// Mitsubishi GX Works2 project: main   PLC: FX3U/FX3UC

PROGRAM MAIN
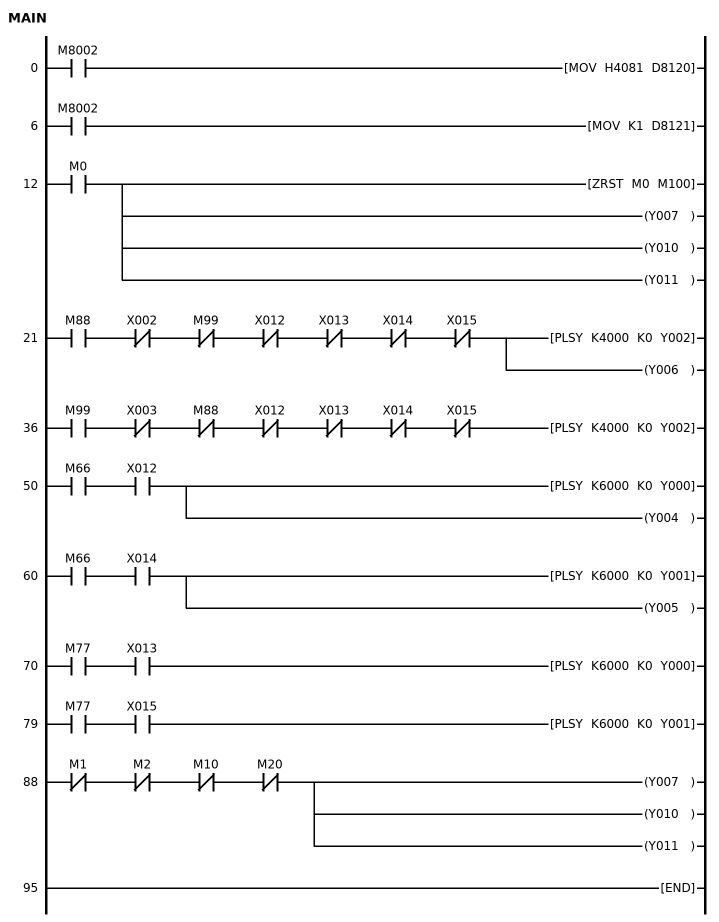
0     LD      M8002
      MOV     H4081 D8120
6     LD      M8002
      MOV     K1 D8121
12    LD      M0
      ZRST    M0 M100
      OUT     Y007
      OUT     Y010
      OUT     Y011
21    LD      M88
      ANI     X002
      ANI     M99
      ANI     X012
      ANI     X013
      ANI     X014
      ANI     X015
      PLSY    K4000 K0 Y002
      OUT     Y006
36    LD      M99
      ANI     X003
      ANI     M88
      ANI     X012
      ANI     X013
      ANI     X014
      ANI     X015
      PLSY    K4000 K0 Y002
50    LD      M66
      AND     X012
      PLSY    K6000 K0 Y000
      OUT     Y004
60    LD      M66
      AND     X014
      PLSY    K6000 K0 Y001
      OUT     Y005
70    LD      M77
      AND     X013
      PLSY    K6000 K0 Y000
79    LD      M77
      AND     X015
      PLSY    K6000 K0 Y001
88    LDI     M1
      ANI     M2
      ANI     M10
      ANI     M20
      OUT     Y007
      OUT     Y010
      OUT     Y011
95    END
END_PROGRAM
